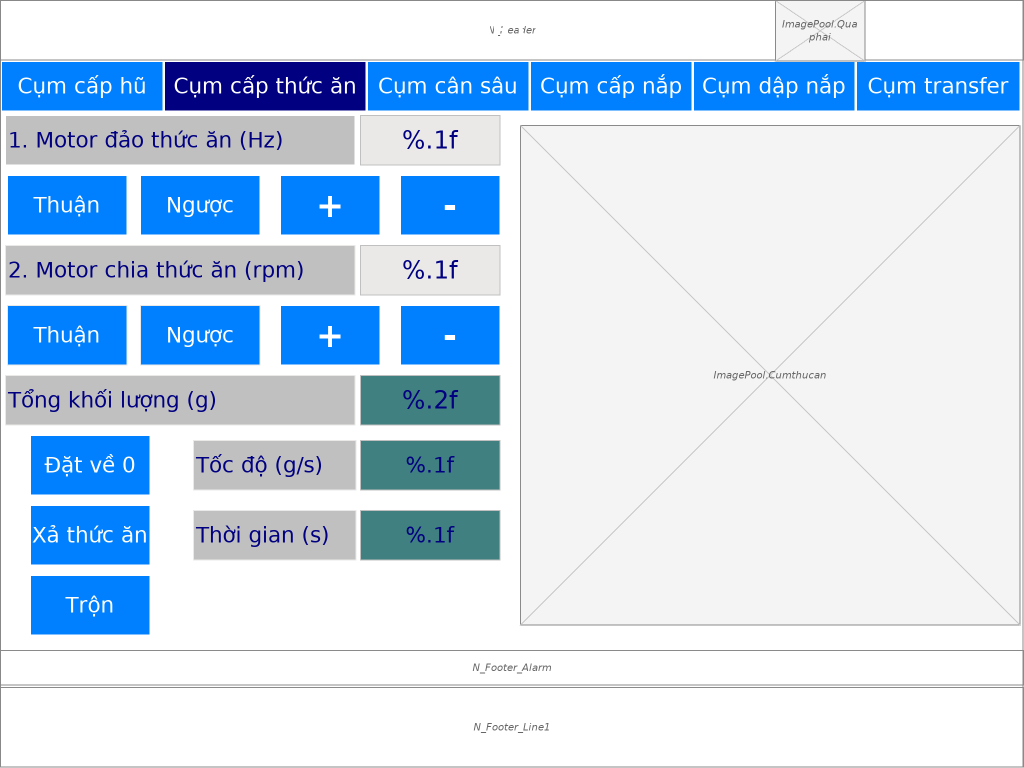
VISUALIZATION N_FoodSupply1  // 1024x768
    Rectangle (30,575 120x60), "Dừng", invisible if: not PR_Line01.daothucan, input disabled if: not PR_Line01.daothucan
        OnMouseDown: execute { PR_Line01.daothucan := FALSE; PR_Line01.bxa := true; }
    Rectangle (30,575 120x60), "Trộn", invisible if: PR_Line01.daothucan, input disabled if: PR_Line01.daothucan
        OnMouseDown: execute { PR_Line01.daothucan := TRUE; PR_Line01.bxa := TRUE; }
    Rectangle (140,175 120x60), "Dừng", invisible if: not PR_Line01.bMotor_mixer_reverse, input disabled if: not PR_Line01.bMotor_mixer_reverse
        OnMouseDown: execute { PR_Line01.bMotor_mixer_reverse := FALSE; }
    Rectangle (140,305 120x60), "Dừng", invisible if: not PR_Line01.bMotor_Food_reverse, input disabled if: not PR_Line01.bMotor_Food_reverse
        OnMouseDown: execute { PR_Line01.bMotor_Food_reverse := FALSE; PR_Line01.bxa := FALSE; }
    Rectangle (140,305 120x60), "Ngược", invisible if: PR_Line01.bMotor_Food_reverse, input disabled if: PR_Line01.bMotor_Food
        OnMouseDown: execute { PR_Line01.bMotor_Food_reverse := TRUE; PR_Line01.bxa := false; }
    Rectangle (140,175 120x60), "Ngược", invisible if: PR_Line01.bMotor_mixer_reverse, input disabled if: PR_Line01.bMotor_mixer_Manual
        OnMouseDown: execute { PR_Line01.bMotor_mixer_reverse := TRUE; PR_Line01.bxa := false; }
    Rectangle (7,305 120x60), "Dừng", invisible if: not PR_Line01.bMotor_Food, input disabled if: not PR_Line01.bMotor_Food
        OnMouseDown: execute { PR_Line01.bMotor_Food := FALSE; PR_Line01.bxa := FALSE; }
    Rectangle (7,305 120x60), "Thuận", invisible if: PR_Line01.bMotor_Food, input disabled if: PR_Line01.bMotor_Food_reverse
        OnMouseDown: execute { PR_Line01.bMotor_Food := TRUE; PR_Line01.bxa := false; }
    Rectangle (7,175 120x60), "Dừng", invisible if: not PR_Line01.bMotor_mixer_Manual, input disabled if: not PR_Line01.bMotor_mixer_Manual
        OnMouseDown: execute { PR_Line01.bMotor_mixer_Manual := FALSE; }
    Rectangle (7,175 120x60), "Thuận", invisible if: PR_Line01.bMotor_mixer_Manual, input disabled if: PR_Line01.bMotor_mixer_reverse
        OnMouseDown: execute { PR_Line01.bMotor_mixer_Manual := TRUE; PR_Line01.bxa := false; }
    Frame (0,687 1024x80)
        shows N_Footer_Line1()
    Frame (0,0 1024x60)
        shows N_Header()
    Textfield (353,5 400x50), "MÀN HÌNH CHẠY TAY LINE 1"
    Rectangle (5,115 350x50), "1. Motor đảo thức ăn (Hz)"
    Rectangle (5,245 350x50), "2. Motor chia thức ăn (rpm)"
    Rectangle (1,61 162x50), "Cụm cấp hũ"
        OnMouseClick: change screen: N_JarSupply1
    Rectangle (164,61 202x50), "Cụm cấp thức ăn"
        OnMouseClick: change screen: N_FoodSupply1
    Rectangle (367,61 162x50), "Cụm cân sâu"
        OnMouseClick: change screen: N_WormWeight1
    Rectangle (530,61 162x50), "Cụm cấp nắp"
        OnMouseClick: change screen: N_LidSupply1
    Rectangle (693,61 162x50), "Cụm dập nắp"
        OnMouseClick: change screen: N_LidPressing1
    Rectangle (856,61 164x50), "Cụm transfer"
        OnMouseClick: change screen: N_Tranfer1
    Rectangle (360,115 140x50), "%.1f", text variable: PR_Line01.fb_FoodMixer.fSpeed_motor_mixer_Manual
        OnMouseDown: write PR_Line01.fb_FoodMixer.fSpeed_motor_mixer_Manual via VisuDialogs.Numpad
    Rectangle (360,245 140x50), "%.1f", text variable: PR_Line01.fb_FoodWeight.fSpeed_Food_Motor_Manual
        OnMouseDown: write PR_Line01.fb_FoodWeight.fSpeed_Food_Motor_Manual via VisuDialogs.Numpad
    Rectangle (5,375 350x50), "Tổng khối lượng (g)"
    Rectangle (280,175 100x60), "+", colour toggle: PR_Line01.bUp_Motor_Mixer
        OnMouseDown: execute { PR_Line01.bUp_Motor_Mixer := TRUE; PR_Line01.bxa := false; }
    Rectangle (400,175 100x60), "-", colour toggle: PR_Line01.bDown_Motor_Mixer
        OnMouseDown: execute { PR_Line01.bDown_Motor_Mixer := TRUE; PR_Line01.bxa := false; }
    Rectangle (280,305 100x60), "+", colour toggle: PR_Line01.bUp_Food_Motor
        OnMouseDown: execute { PR_Line01.bUp_Food_Motor := TRUE; PR_Line01.bxa := FALSE; }
    Rectangle (400,305 100x60), "-", colour toggle: PR_Line01.bDown_Food_Motor
        OnMouseDown: execute { PR_Line01.bDown_Food_Motor := TRUE; PR_Line01.bxa := false; }
    Rectangle (360,375 140x50), "%.2f", text variable: PR_Line01.fb_FoodWeight.fWeight_Food
    Rectangle (193,440 163x50), "Tốc độ (g/s)"
    Rectangle (360,440 140x50), "%.1f", text variable: PR_Line01.fb_FoodWeight.fFlow_Food
    Image (775,0 90x61), input disabled if: bResetAuto2, image: ImagePool.Qua phai
        OnMouseClick: change screen: N_FoodSupply2
        OnMouseClick: execute { MAIN_LINE2.bModeManual := TRUE; MAIN_LINE2.bModeAuto := FALSE; }
    Rectangle (30,435 120x60), "Đặt về 0", colour toggle: PR_Line01.bZero_Loadcell_Food
        tap PR_Line01.bZero_Loadcell_Food
        OnMouseDown: execute { PR_Line01.bxa := false; }
        OnMouseUp: execute { PR_Line01.bZero_Loadcell_Food := TRUE; }
    Rectangle (30,505 120x60), "Xả thức ăn", colour toggle: PR_Line01.xathucan
        OnMouseDown: execute { PR_Line01.xathucan := TRUE; PR_Line01.bxa := TRUE; }
    Rectangle (193,510 163x50), "Thời gian (s)"
    Rectangle (360,510 140x50), "%.1f", text variable: PR_Line01.fb_FoodWeight.fTime
    Image (520,125 500x500), image: ImagePool.Cumthucan
    Frame (0,650 1024x35)
        shows N_Footer_Alarm()
END_VISUALIZATION

(* stored: Version 1.1.0.1, ProductVersion 3.1.4024.12
   Visu N_FoodSupply1: Id {889aa8d6-5cdc-4254-bc90-b371095acb51} *)
